PROGRAM POU_Example
VAR
END_VAR

(* Here we call all the function block that have been declared in GVL_Devices*)


//Pirani Gauges
FEE_GPI_01();
FEE_GPI_02(PG=>);
// Ion Gauges
FEE_GCC_01(PG:= FEE_GPI_01.PG);
FEE_GCC_02(PG:= FEE_GPI_02.PG, IG=>);

//Isolation Valves
FEE_VGC_01(i_stUSG := FEE_GCC_01.IG, i_stDSG := FEE_GCC_02.IG, i_xDis_DPIlk:=TRUE, i_xEPS_OK:= TRUE, i_xPMPS_OK :=TRUE);

//Ion Pumps

END_PROGRAM

(* stored: Version 1.1.0.1, ProductVersion 3.1.4022.12
   POU POU_Example: Id {5d330a11-7bbf-4631-b77e-0e51d0207e45}, SpecialFunc None *)
